FUNCTION_BLOCK FEATURE_EXTRACTION
  {SET_ATTRIBUTE(OpcUa, SERVICE)}
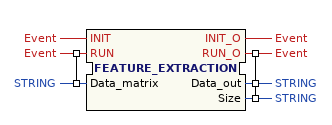
  EVENT_INPUT
    INIT;
    RUN WITH Data_matrix; {SET_ATTRIBUTE(OpcUa, Method)}
  END_EVENT
  EVENT_OUTPUT
    INIT_O;
    RUN_O WITH Data_out, Size;
  END_EVENT
  VAR_INPUT
    Data_matrix : STRING; {SET_ATTRIBUTE(OpcUa, Variable.RUN)}
  END_VAR
  VAR_OUTPUT
    Data_out : STRING; {SET_ATTRIBUTE(OpcUa, Variable.RUN)}
    Size : STRING; {SET_ATTRIBUTE(OpcUa, Variable.RUN)}
  END_VAR
END_FUNCTION_BLOCK
